// TIA Portal V21 export
FUNCTION_BLOCK "FB1"   // FB8, LAD
{ S7_Optimized_Access := 'FALSE' }
// stored: AutoNumber false, SetENOAutomatically false
   VAR_INPUT
      TIME_START : Bool;
      TIME_PULSE : Bool;
      TIME_TRSET : Bool;
      MINI_ENABLE : Bool;
      TIME_IN_MINI : Int;
      TIME_IN_SEC : Int;
   END_VAR
   VAR_OUTPUT
      DONE_BIT : Bool;
      ES_MINIT : DInt;
      ES_SEC : DInt;
   END_VAR
   VAR_IN_OUT
      TEMP_1 : Int;
      TEMP_5 : Int;
      TEMP_2 : Int;
      TEMP_3 : Int;
      TEMP_4 : DInt;
      TEMP_BIT_1 : Bool;
   END_VAR
BEGIN

REGION Network 1
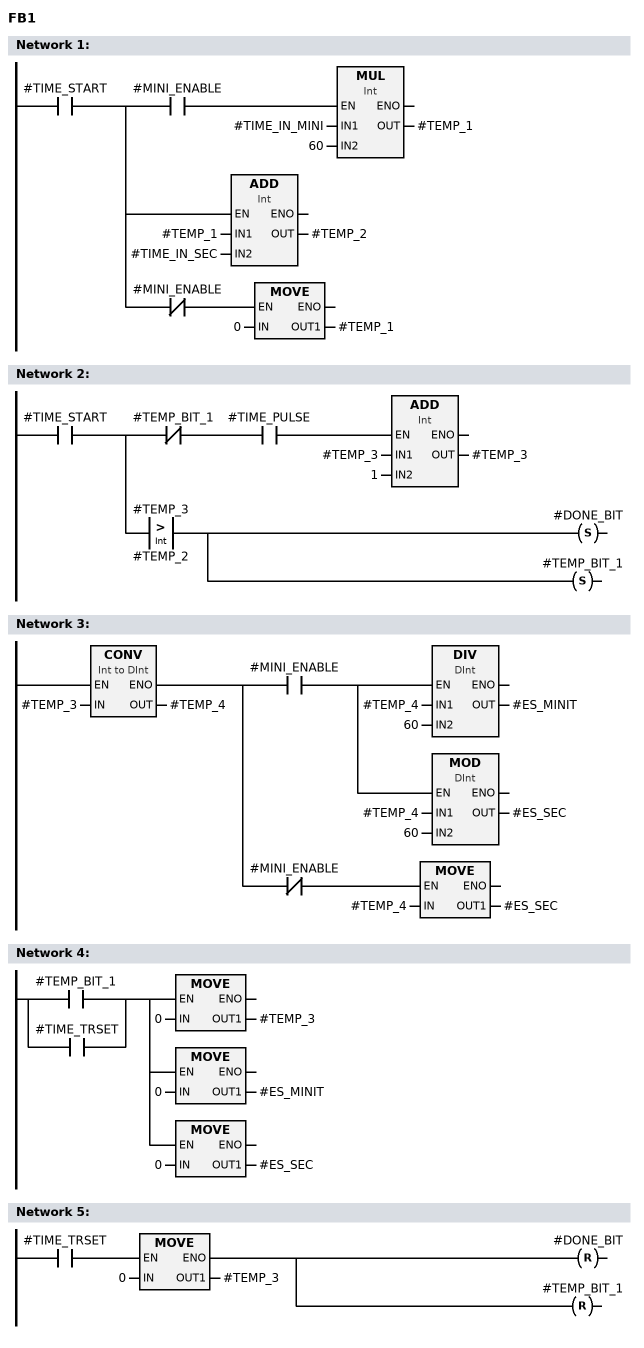
   RUNG wire#powerrail
      Contact( #TIME_START )
      wire#w1
      Contact( #MINI_ENABLE )
      { S7_Templates := "SrcType := Int"; S7_GenerateENO := "TRUE" } Mul(in1 := #TIME_IN_MINI, in2 := 60, out => #TEMP_1)
   END_RUNG
   RUNG wire#w1
      { S7_Templates := "SrcType := Int"; S7_GenerateENO := "TRUE" } Add(in1 := #TEMP_1, in2 := #TIME_IN_SEC, out => #TEMP_2)
   END_RUNG
   RUNG wire#w1
      I_Contact( #MINI_ENABLE )
      { S7_GenerateENO := "TRUE" } Move(in := 0, out1 => #TEMP_1)
   END_RUNG
   // the same network as SCL:
   IF #TIME_START AND #MINI_ENABLE THEN #TEMP_1 := #TIME_IN_MINI * 60; END_IF;
   IF #TIME_START THEN #TEMP_2 := #TEMP_1 + #TIME_IN_SEC; END_IF;
   IF #TIME_START AND NOT #MINI_ENABLE THEN #TEMP_1 := 0; END_IF;
END_REGION

REGION Network 2
   RUNG wire#powerrail
      Contact( #TIME_START )
      wire#w1
      I_Contact( #TEMP_BIT_1 )
      Contact( #TIME_PULSE )
      { S7_Templates := "SrcType := Int"; S7_GenerateENO := "TRUE" } Add(in1 := #TEMP_3, in2 := 1, out => #TEMP_3)
   END_RUNG
   RUNG wire#w1
      { S7_Templates := "SrcType := Int" } GT_Contact(in1 := #TEMP_3, in2 := #TEMP_2)
      wire#w2
      S_Coil( #DONE_BIT )
   END_RUNG
   RUNG wire#w2
      S_Coil( #TEMP_BIT_1 )
   END_RUNG
   // the same network as SCL:
   IF #TIME_START AND NOT #TEMP_BIT_1 AND #TIME_PULSE THEN #TEMP_3 := #TEMP_3 + 1; END_IF;
   IF #TIME_START AND (#TEMP_3 > #TEMP_2) THEN
       #DONE_BIT := TRUE;
       #TEMP_BIT_1 := TRUE;
   END_IF;
END_REGION

REGION Network 3
   RUNG wire#powerrail
      { S7_Templates := "[SrcType := Int, DestType := DInt]"; S7_GenerateENO := "TRUE" } Convert(in := #TEMP_3, out => #TEMP_4)
      wire#w1
      Contact( #MINI_ENABLE )
      wire#w2
      { S7_Templates := "SrcType := DInt"; S7_GenerateENO := "TRUE" } Div(in1 := #TEMP_4, in2 := 60, out => #ES_MINIT)
   END_RUNG
   RUNG wire#w2
      { S7_Templates := "SrcType := DInt"; S7_GenerateENO := "TRUE" } Mod(in1 := #TEMP_4, in2 := 60, out => #ES_SEC)
   END_RUNG
   RUNG wire#w1
      I_Contact( #MINI_ENABLE )
      { S7_GenerateENO := "TRUE" } Move(in := #TEMP_4, out1 => #ES_SEC)
   END_RUNG
   // the same network as SCL:
   // ENO of a box is taken as its EN; it also drops when the box reports an error
   #TEMP_4 := INT_TO_DINT(#TEMP_3);
   IF #MINI_ENABLE THEN
       #ES_MINIT := #TEMP_4 / 60;
       #ES_SEC := #TEMP_4 MOD 60;
   END_IF;
   IF NOT #MINI_ENABLE THEN #ES_SEC := #TEMP_4; END_IF;
END_REGION

REGION Network 4
   RUNG wire#powerrail
      Contact( #TEMP_BIT_1 )
      wire#w1
      { S7_GenerateENO := "TRUE" } Move(in := 0, out1 => #TEMP_3)
   END_RUNG
   RUNG wire#powerrail
      Contact( #TIME_TRSET )
   END_RUNG wire#w1
   RUNG wire#w1
      { S7_GenerateENO := "TRUE" } Move(in := 0, out1 => #ES_MINIT)
   END_RUNG
   RUNG wire#w1
      { S7_GenerateENO := "TRUE" } Move(in := 0, out1 => #ES_SEC)
   END_RUNG
   // the same network as SCL:
   IF #TEMP_BIT_1 OR #TIME_TRSET THEN
       #TEMP_3 := 0;
       #ES_MINIT := 0;
       #ES_SEC := 0;
   END_IF;
END_REGION

REGION Network 5
   RUNG wire#powerrail
      Contact( #TIME_TRSET )
      { S7_GenerateENO := "TRUE" } Move(in := 0, out1 => #TEMP_3)
      wire#w1
      R_Coil( #DONE_BIT )
   END_RUNG
   RUNG wire#w1
      R_Coil( #TEMP_BIT_1 )
   END_RUNG
   // the same network as SCL:
   // ENO of a box is taken as its EN; it also drops when the box reports an error
   IF #TIME_TRSET THEN
       #TEMP_3 := 0;
       #DONE_BIT := FALSE;
       #TEMP_BIT_1 := FALSE;
   END_IF;
END_REGION
END_FUNCTION_BLOCK
